{attribute 'linkalways'} 
{attribute 'no_explicit_call' := 'This FB is a CLASS and must be accessed using methods or properties'}
{attribute 'enable_dynamic_creation'}
FUNCTION_BLOCK Node_F_VN_DistanceTransformation EXTENDS VisionNode
VAR
    ipSrcImage : _ITcVnImage;
    ipDestImage : _ITcVnImage;
    eDistanceType : _ETcVnDistanceType(ETcVnDistanceType.TCVN_DT_L1);
    eMaskSize : _ETcVnDistanceTransformationMask(ETcVnDistanceTransformationMask.TCVN_DTM_PRECISE);
    hrPrev : _HRESULT(S_OK);
	hresult : _HRESULT(S_OK);
END_VAR

METHOD PUBLIC  Clone : I_Node
VAR
	pNode : POINTER TO Node_F_VN_DistanceTransformation;
END_VAR
pNode := __NEW(Node_F_VN_DistanceTransformation);
Clone := pNode^;
END_METHOD

METHOD FB_init : BOOL
VAR_INPUT
	bInitRetains : BOOL; // if TRUE, the retain variables are initialized (warm start / cold start)
	bInCopyCode : BOOL;  // if TRUE, the instance afterwards gets moved into the copy code (online change)
END_VAR
AddInput('ipSrcImage', ipSrcImage);
AddParameter('eDistanceType', eDistanceType);
AddParameter('eMaskSize', eMaskSize);
AddInput('hrPrev', hrPrev);
AddOutput('ipDestImage', ipDestImage);
AddOutput('hresult',hresult);
END_METHOD

METHOD PROTECTED OnExecute
hresult.Value := F_VN_DistanceTransformation(
    ipSrcImage := ipSrcImage.Value,
	ipDestImage := ipDestImage.Value,
    eDistanceType := eDistanceType.Value,
    eMaskSize := eMaskSize.Value,
	hrPrev:= hrPrev.Value);
END_METHOD

METHOD PUBLIC PreExecutionCheck
VAR_INPUT
	Check : I_PreExecutionChecks;
END_VAR
VAR
    distanceTypeIsValid : BOOL;
END_VAR
Check.IsTrue(ipSrcImage.IsValid, 'ipSrcImage must contain an image');
Check.IsTrue(ipSrcImage.HasChannelCount(1), 'ipSrcImage must have 1 channel');
Check.IsTrue(ipSrcImage.IsPixelDepth(8), 'ipSrcImage must have 8 bit pixel depth');

CASE eDistanceType.Value OF
    ETcVnDistanceType.TCVN_DT_L1,
    ETcVnDistanceType.TCVN_DT_L2,
    ETcVnDistanceType.TCVN_DT_C :
        distanceTypeIsValid := TRUE;
END_CASE
Check.IsTrue(distanceTypeIsValid, 'eDistanceType value is unsupported');
END_METHOD

END_FUNCTION_BLOCK

(* stored: Version 1.1.0.1, ProductVersion 3.1.4024.15
   POU Node_F_VN_DistanceTransformation: Id {4d91cd47-be3b-0012-3a2c-291becfd9006}, SpecialFunc None
   Folder Constructor: Id {9681b2ee-e1a0-050e-2bfe-ad775bdee409}
   Method Clone: Id {538efdff-d2ce-0e11-071b-fad8805e1b16}
   Method FB_init: Id {8f56763e-b312-08a0-0925-73f227f64a0f}
   Method OnExecute: Id {843db459-d414-0e20-2692-b339d34691ef}
   Method PreExecutionCheck: Id {0105c7e8-4618-0920-3bb3-8df9736f5174} *)
